FUNCTION F_GetFunctionSettings : ST_CFG_Function
(**************************************************************************************
 * 	Application		:	BoxControl Framework
 *	Revision		:	$Revision: 404529 $
 *	Revision date	:	$Date: 2018-04-23 08:21:38 +0200 (Mo., 23 Apr 2018) $
 *	Last changed by	:	$Author: b7bolm $
 *	URL				:	$URL: http://almscdc.swisslog.com/repo/SWPD/Development/BoxControlFramework/20_Release/trunk/01_Software/BCF/BCF/JumpStart/20_Product/10_App/12_E_Functions/10_Lib/10_Conv/10_Functions/F_GetFunctionSettings.TcPOU $
 *
 *	Purpose			:	Function settings.
 *
 * ------------------------------------------------------------------------------------
 *	Copyright Swisslog [IP AG], Switzerland. All rights reserved.
 * 
 * ------------------------------------------------------------------------------------
 *	
 * 	Revision History: 
 *
 * 	VERSION			DATE			INITIALS			DESCRIPTION
 *	0.1				01.01.2001		swl					Example
 *
 **************************************************************************************)
VAR_INPUT
	eFunctionNumber		: E_FunctionNumber; // Function number
END_VAR

// If reference is valid
IF __ISVALIDREF(FunctionRegistry[eFunctionNumber].rSettingsFunction) THEN
	// Return base settings
	F_GetFunctionSettings := FunctionRegistry[eFunctionNumber].rSettingsFunction;
END_IF

END_FUNCTION

(* stored: Version 1.1.0.1, ProductVersion 3.1.4022.12
   POU F_GetFunctionSettings: Id {d1cae01d-f948-4c5d-9982-a8a51083d004}, SpecialFunc None *)
